(* PLC project Unnamed, Unknown Unnamed 1 *)
(* stored: creationDateTime 2024-09-04T10:51:37, modificationDateTime 2024-11-07T14:10:11 *)

PROGRAM lift
  VAR
    assigned_pallet_rack : SINT := 6;
    lift_up_motor : BOOL;
    lift_down_motor : BOOL;
    conveyor_motor : BOOL;
    current_rack : SINT := 0;
    initial_rack : SINT := 0;
    TON0 : TON;
    TON1 : TON;
  END_VAR
  VAR  (* added by the conversion: wires and edge detectors of the diagram *)
    _GT5_OUT : BOOL;
    _EQ12_OUT : BOOL;
    _EQ23_OUT : BOOL;
  END_VAR

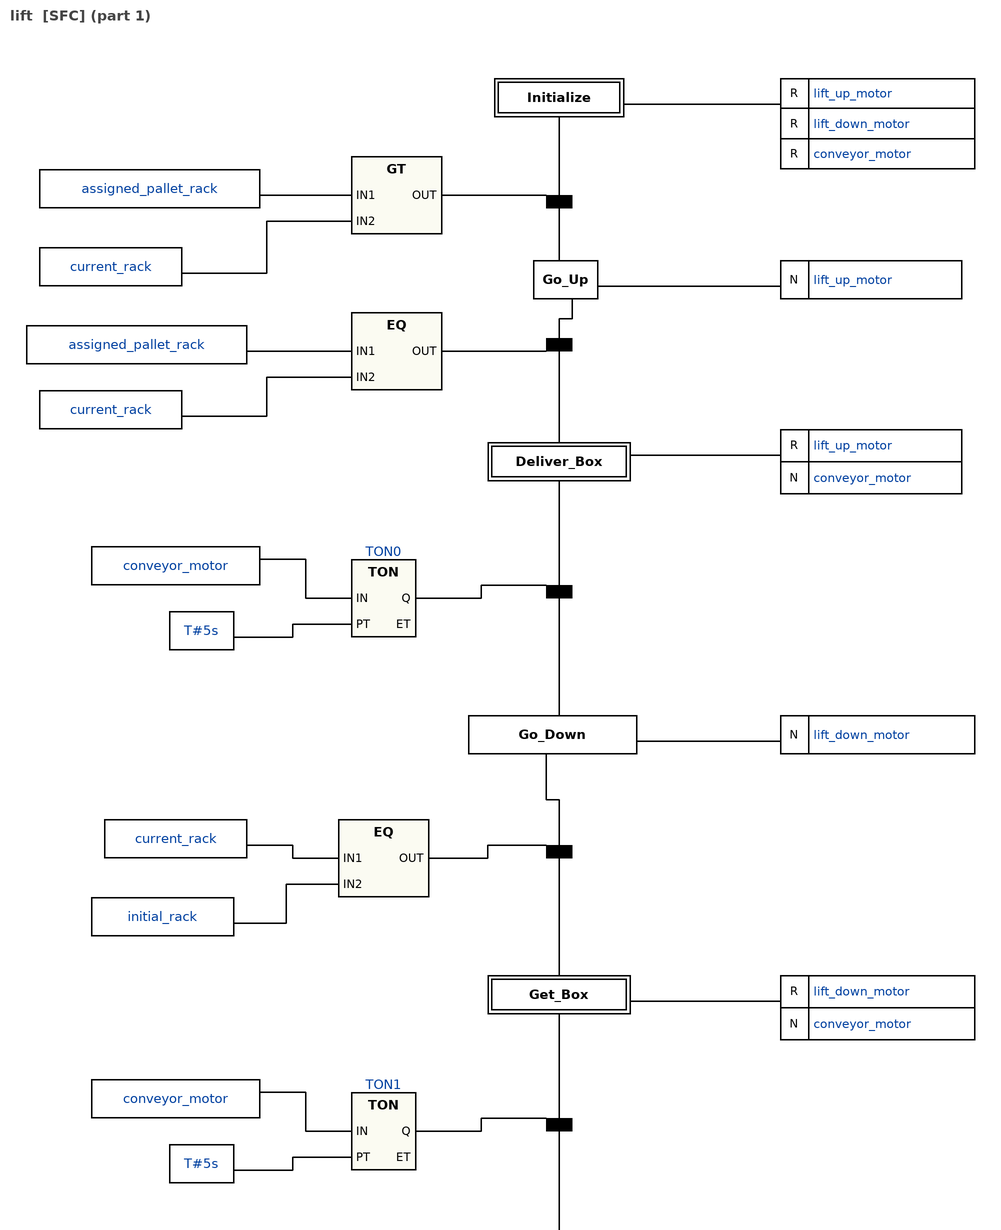
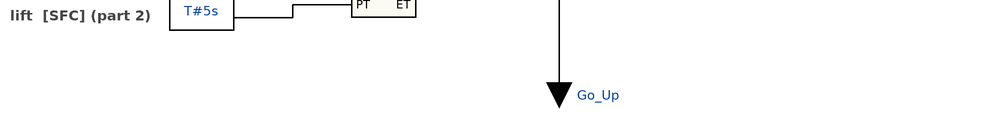
INITIAL_STEP Initialize:
  lift_up_motor(R);
  lift_down_motor(R);
  conveyor_motor(R);
  COMPUTE_FUNCTION_BLOCKS(S);
END_STEP
TRANSITION FROM Initialize TO Go_Up
  := _GT5_OUT;
END_TRANSITION
INITIAL_STEP Deliver_Box:
  lift_up_motor(R);
  conveyor_motor(N);
END_STEP
TRANSITION FROM Deliver_Box TO Go_Down
  := TON0.Q;
END_TRANSITION
INITIAL_STEP Get_Box:
  lift_down_motor(R);
  conveyor_motor(N);
END_STEP
TRANSITION FROM Get_Box TO Go_Up
  := TON1.Q;
END_TRANSITION
STEP Go_Up:
  lift_up_motor(N);
END_STEP
TRANSITION FROM Go_Up TO Deliver_Box
  := _EQ12_OUT;
END_TRANSITION
STEP Go_Down:
  lift_down_motor(N);
END_STEP
TRANSITION FROM Go_Down TO Get_Box
  := _EQ23_OUT;
END_TRANSITION
ACTION COMPUTE_FUNCTION_BLOCKS:  (* blocks drawn on the SFC sheet *)
  _GT5_OUT := assigned_pallet_rack > current_rack;
  TON0(IN := conveyor_motor, PT := T#5s);
  TON1(IN := conveyor_motor, PT := T#5s);
  _EQ12_OUT := assigned_pallet_rack = current_rack;
  _EQ23_OUT := current_rack = initial_rack;
END_ACTION
END_PROGRAM

CONFIGURATION Config0
  RESOURCE Res0 ON PLC
    TASK task0(INTERVAL := T#20ms, PRIORITY := 0);
    PROGRAM instance0 WITH task0 : lift;
  END_RESOURCE
END_CONFIGURATION
